PROGRAM state_transition
VAR PERSISTENT
END_VAR

// NETWORK 1

END_PROGRAM

(* stored: Version 1.1.0.1, ProductVersion 3.1.4024.12
   POU state_transition: Id {48687b9f-7057-49bd-b80e-9cc206fe590e}, SpecialFunc None *)
